(* PLC project Unnamed, Unknown Unnamed 1 *)
(* stored: creationDateTime 2026-03-21T21:56:53, modificationDateTime 2026-03-21T22:24:29 *)

PROGRAM E8
  VAR
    TON0 : TON;
    TON1 : TON;
  END_VAR
  VAR_INPUT
    S_MILL : BOOL;
    S_DRILL : BOOL;
  END_VAR
  VAR_OUTPUT
    CV1 : BOOL;
    CV2 : BOOL;
    CV3 : BOOL;
  END_VAR
  VAR_INPUT
    CV4 : BOOL;
  END_VAR
  VAR
    M_RUN : BOOL;
    M_MILLING : BOOL;
    M_TO_DRILL : BOOL;
    M_DRILLING : BOOL;
    M_TO_EXIT : BOOL;
  END_VAR

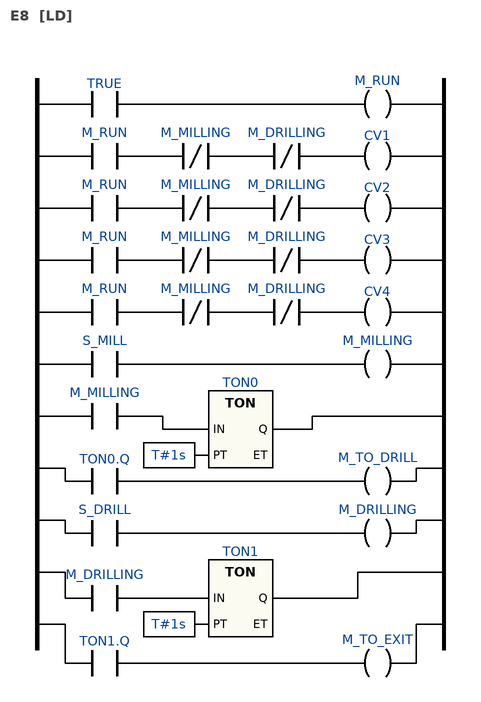
(* LD diagram, written out as Structured Text *)
M_RUN := TRUE;
CV1 := M_RUN AND NOT M_MILLING AND NOT M_DRILLING;
CV2 := M_RUN AND NOT M_MILLING AND NOT M_DRILLING;
CV3 := M_RUN AND NOT M_MILLING AND NOT M_DRILLING;
CV4 := M_RUN AND NOT M_MILLING AND NOT M_DRILLING;
M_MILLING := S_MILL;
M_TO_DRILL := TON0.Q;
M_DRILLING := S_DRILL;
M_TO_EXIT := TON1.Q;
TON0(IN := M_MILLING, PT := T#1s);
TON1(IN := M_DRILLING, PT := T#1s);
END_PROGRAM

CONFIGURATION Config0
  RESOURCE Res0 ON PLC
    TASK task0(INTERVAL := T#20ms, PRIORITY := 0);
    PROGRAM instance0 WITH task0 : E8;
  END_RESOURCE
END_CONFIGURATION
